# EPICS substitutions: iocBoot/iocTomoScan_BEATS_PCO_ACS_Cont/tomoScan.substitutions
file "$(TOP)/db/tomoScan.template"
{
pattern
{P,              R,             CAMERA,    FILE_PLUGIN,    ROTATION, SAMPLE_X, SAMPLE_Y, CLOSE_COMBINED_STOPPER_SHUTTER, CLOSE_VALUE, OPEN_COMBINED_STOPPER_SHUTTER, OPEN_VALUE, COMBINED_STOPPER_SHUTTER_STATUS, CLOSE_VALUE_STATUS, OPEN_VALUE_STATUS, ROT_INTERNAL_MAX_SPEED, ROTARY_PRESSURE_INTERLOCK, X_PRESSURE_INTERLOCK, Y_PRESSURE_INTERLOCK, ROTARY_ENABLED, X_ENABLED, Y_ENABLED, ACS_ENABLE, X_VALVE, Y_VALVE, INTERLOCK_RESET, EMERGENCY_BUTTON}
{tomoscanBEATS:, PcoAcsCont:, TEST-PCO:, TEST-PCO:HDF1:, I10R3-MO-ACS:EH-TMO-SRV-ROT:m1, I10R2-MO-MC2:EH-TMO-STP-TRSX1,   I10R2-MO-MC2:EH-TMO-STP-TRSY1,   I10OH-VA-COMB:setClose,         1,           I10OH-VA-COMB:setOpen,         1,          I10OH-VA-COMB:getStatus, 1,    3, BEATS:RotInt:MaxSpeed.VAL, I10EH-ES-ACS-PRESSURE-R:isOn, I10EH-ES-ACS-CLAMPX:isOn, I10EH-ES-ACS-PRESSURE-Y:isOn, I10EH-ES-ACS-R-MOTOR:isEnabled, I10EH-ES-ACS-X-MOTOR:isEnabled, I10EH-ES-ACS-Y-MOTOR:isEnabled, I10R3-MO-ACS:EH-TMO-SRV-ROT:m1.CNEN, I10EH-ES-ACS-VALVE-X:turnOn, I10EH-ES-ACS-VALVE-Y:turnOff, I10EH-ES-ACS:reset, I10EH-ES-ACS-EM:isPressed}
}

file "$(TOP)/db/tomoScan_BEATS_PCO_ACS_Cont.template"
{
pattern
{P,              R,             BEAM_READY,              READY_VALUE, EXPOSURE_SHUTTER,}
{tomoscanBEATS:, PcoAcsCont:, BEAMREADY:ShutterPermit, 1,           I10EH-SHUTTER:command,}
}
